FUNCTION IO_TO_APT : ST_PMPS_Aperture
VAR_INPUT
    IO : ST_PMPS_Aperture_IO;
END_VAR
VAR
END_VAR

IO_TO_APT.Height := IO.Height;
IO_TO_APT.Width := IO.Width;
IO_TO_APT.xOK := IO.xOK;

END_FUNCTION

(* stored: Version 1.1.0.1
   POU IO_TO_APT: Id {612c94fe-4ac7-47d4-a1e8-700a8f5271ed}, SpecialFunc None *)
